(* PLC project Unnamed, Unknown Unnamed 1 *)
(* stored: creationDateTime 2024-01-09T16:45:07, modificationDateTime 2024-01-23T14:31:54 *)

CONFIGURATION config
  RESOURCE resource1 ON PLC
    TASK task0(INTERVAL := T#20ms, PRIORITY := 0);
    PROGRAM instance0 WITH task0 : {{ programs[0] }};
  END_RESOURCE
END_CONFIGURATION
